// TIA Portal V20 export
TYPE "LER_typeCommunicationBRCVParameter"
// stored: Access Published
   STRUCT
      Input : Struct
         EN_R : Bool;
      END_STRUCT;
      Output : Struct
         len : Word;
         ndr : Bool;
         error : Bool;
         status : Word;
      END_STRUCT;
   END_STRUCT;
END_TYPE
